PROGRAM IO
VAR
END_VAR

(*
 NAME:		16435-MOBILEHOIST
 CREATED:	10/30/2022 
 AUTHOR:	RRODRIGUEZ-HERNANDEZ
 FIRST PROTOTYPE
*)

(*INPUTS - CX8190-EL1859-1*)
MOBILEHOIST.SYSTEM_RESET					:=INPUT.EL1859_1.0;						//INPUT 1
MOBILEHOIST.ESTOP_CONDITION					:=INPUT.EL1859_1.1 = FALSE;				//INPUT 2
MOBILEHOIST.FLOORPOSITION_SWITCH1			:=INPUT.EL1859_1.2;						//INPUT 3
MOBILEHOIST.FLOORPOSITION_SWITCH2			:=INPUT.EL1859_1.3;						//INPUT 4
MOBILEHOIST.TEMP_SWITCH						:=INPUT.EL1859_1.4;						//INPUT 5
MOBILEHOIST.DEADMAN_SWITCH					:=INPUT.EL1859_1.5;						//INPUT 6

(*OUTPUTS - CX8190-EL1859-1*)
OUTPUT.EL1859_1.0 							:=MOBILEHOIST.RESETPB_LED;				//OUTPUT 1			
OUTPUT.EL1859_1.1                           :=MOBILEHOIST.SELECTORSW_LED;			//OUTPUT 2									
OUTPUT.EL1859_1.2                           :=MOBILEHOIST.MAGNETIC_BRAKE1;			//OUTPUT 3
OUTPUT.EL1859_1.3 							:=MOBILEHOIST.MAGNETIC_BRAKE2;			//OUTPUT 4			
OUTPUT.EL1859_1.4                           :=MOBILEHOIST.MAINPWR;					//OUTPUT 5
OUTPUT.EL1859_1.4                           :=MOBILEHOIST.SPOTLIGHT;				//OUTPUT 6

(*OUTPUTS - CX8190-EL1859-2*)
OUTPUT.EL1859_2.0 							:=MOBILEHOIST.REDSTACKLIGHT;			//OUTPUT 1			
OUTPUT.EL1859_2.1                           :=MOBILEHOIST.AMBERSTACKLIGHT;			//OUTPUT 2		

(*STATE*)
MOBILEHOIST.IOSTATE1						:=INPUT.EL1859_1_STATE.3;
MOBILEHOIST.IOSTATE2						:=INPUT.EL1859_2_STATE.3;

END_PROGRAM

(* stored: Version 1.1.0.1, ProductVersion 3.1.4024.11
   POU IO: Id {c5b9e636-c88d-49e4-9b5d-fe919b6a53df}, SpecialFunc None *)
